{attribute 'GeneratedUsingTerminal: EPP1258-0001-0016'}
{attribute addProperty BoxType "EPP1258-0001-0016"}
{attribute addProperty Id "Status0AT %I*USINT1Status1AT %I*USINT1LatchPos0AT %I*ULINT8LatchNeg0AT %I*ULINT8LatchPos1AT %I*ULINT8LatchNeg1AT %I*ULINT8"}
{attribute addProperty CRC "2386637461"}
{attribute addProperty Size "34"}
TYPE Latch_8E413295 EXTENDS InputBase_8311D824 :
STRUCT
	{attribute addProperty Name "Status0"}
	Status0 AT %I* : USINT;
	{attribute addProperty Name "Status1"}
	Status1 AT %I* : USINT;
	{attribute addProperty Name "LatchPos0"}
	LatchPos0 AT %I* : ULINT;
	{attribute addProperty Name "LatchNeg0"}
	LatchNeg0 AT %I* : ULINT;
	{attribute addProperty Name "LatchPos1"}
	LatchPos1 AT %I* : ULINT;
	{attribute addProperty Name "LatchNeg1"}
	LatchNeg1 AT %I* : ULINT;
END_STRUCT
END_TYPE

(* stored: Version 1.2.0.0, ProductVersion 3.1.4024.11
   DUT Latch_8E413295: Id {883b644b-943a-4079-837e-40846b56d407} *)
